// TIA Portal V17 export
// export: Created 2022-07-28T18:03:03.6138582Z, ExportSetting None, DisplayName Totally Integrated Automation Portal, DisplayVersion V17, DisplayName TIA Portal Openness, DisplayVersion V17, DisplayName TIA Portal Teamcenter Gateway, DisplayVersion V17, DisplayName TIA Portal Version Control Interface, DisplayVersion V17, DisplayName TIA Portal Test Suite Advanced, DisplayVersion V17, DisplayName SINAMICS Startdrive Advanced, DisplayVersion V17, DisplayName SINAMICS DCC, DisplayVersion V17, DisplayName SINAMICS Startdrive G130, G150, S120, S150, SINAMICS MV, S210, DisplayVersion V17, DisplayName SINAMICS Startdrive G110M, G120, G120C, G120D, G120P, G115D, DisplayVersion V17, DisplayName STEP 7 Professional, DisplayVersion V17, DisplayName SIMATIC Energy Suite, DisplayVersion V17, DisplayName STEP 7 CFC, DisplayVersion V17, DisplayName STEP 7 Safety, DisplayVersion V17, DisplayName WinCC Advanced / Unified PC, DisplayVersion V17, DisplayName SIMATIC Visualization Architect, DisplayVersion V17
DATA_BLOCK "D_ZeroTypes"   // DB5
{ S7_Optimized_Access := 'TRUE' }
// stored: IsWriteProtectedInAS true, MemoryReserve 100
   VAR
      ASensor_HMI { ExternalAccessible := 'False'; ExternalVisible := 'False'; ExternalWritable := 'False'} : "lib_udt_ASensor_HMI";
      ASensor_PLC { ExternalAccessible := 'False'; ExternalVisible := 'False'; ExternalWritable := 'False'} : "lib_udt_ASensor_PLC";
      AnalogFlowmeter_HMI { ExternalAccessible := 'False'; ExternalVisible := 'False'; ExternalWritable := 'False'} : "lib_udt_AnalogFlowmeter_HMI";
      AnalogFlowmeter_PLC { ExternalAccessible := 'False'; ExternalVisible := 'False'; ExternalWritable := 'False'} : "lib_udt_AnalogFlowmeter_PLC";
      DSensor_HMI { ExternalAccessible := 'False'; ExternalVisible := 'False'; ExternalWritable := 'False'} : "lib_udt_DSensor_HMI";
      DSensor_PLC { ExternalAccessible := 'False'; ExternalVisible := 'False'; ExternalWritable := 'False'} : "lib_udt_DSensor_PLC";
      Inverter_352Tel { ExternalAccessible := 'False'; ExternalVisible := 'False'; ExternalWritable := 'False'} : "Lib_UDT_Inverter_352Tel";
      SlideGate_Pneumo_PLC { ExternalAccessible := 'False'; ExternalVisible := 'False'; ExternalWritable := 'False'} : "Lib_UDT_SlideGate_Pneumo_PLC";
      SlideGate_Pneumo_HMI { ExternalAccessible := 'False'; ExternalVisible := 'False'; ExternalWritable := 'False'} : "Lib_UDT_SlideGate_Pneumo_HMI";
      Pump_Inv352_Base_HMI { ExternalAccessible := 'False'; ExternalVisible := 'False'; ExternalWritable := 'False'} : "Lib_UDT_Pump_Inv352_Base_HMI";
      Pump_Inv352_Base_PLC { ExternalAccessible := 'False'; ExternalVisible := 'False'; ExternalWritable := 'False'} : "Lib_UDT_Pump_Inv352_Base_PLC";
      Pump_DS_Base_HMI { ExternalAccessible := 'False'; ExternalVisible := 'False'; ExternalWritable := 'False'} : "Lib_UDT_Pump_DS_Base_HMI";
      Pump_DS_Base_PLC { ExternalAccessible := 'False'; ExternalVisible := 'False'; ExternalWritable := 'False'} : "Lib_UDT_Pump_DS_Base_PLC";
      PID_Base_HMI { ExternalAccessible := 'False'; ExternalVisible := 'False'; ExternalWritable := 'False'} : "Lib_UDT_PID_Base_HMI";
      PID_Base_PLC { ExternalAccessible := 'False'; ExternalVisible := 'False'; ExternalWritable := 'False'} : "Lib_UDT_PID_Base_PLC";
      PID_Cascad_HMI { ExternalAccessible := 'False'; ExternalVisible := 'False'; ExternalWritable := 'False'} : "Lib_UDT_PID_Cascad_HMI";
      PID_Cascad_PLC { ExternalAccessible := 'False'; ExternalVisible := 'False'; ExternalWritable := 'False'} : "Lib_UDT_PID_Cascad_PLC";
      PID_Core { ExternalAccessible := 'False'; ExternalVisible := 'False'; ExternalWritable := 'False'} : "Lib_UDT_PID_Core";
      SlideGate_Cond_PLC { ExternalAccessible := 'False'; ExternalVisible := 'False'; ExternalWritable := 'False'} : "Lib_UDT_SlideGate_Cond_PLC";
      SlideGate_Cond_HMI { ExternalAccessible := 'False'; ExternalVisible := 'False'; ExternalWritable := 'False'} : "Lib_UDT_SlideGate_Cond_HMI";
      SlideGate_Blow_PLC { ExternalAccessible := 'False'; ExternalVisible := 'False'; ExternalWritable := 'False'} : "Lib_UDT_SlideGate_Blow_PLC";
      SlideGate_Blow_HMI { ExternalAccessible := 'False'; ExternalVisible := 'False'; ExternalWritable := 'False'} : "Lib_UDT_SlideGate_Blow_HMI";
   END_VAR
BEGIN
END_DATA_BLOCK
